INTERFACE ITF_BaseHMIComponent_View EXTENDS ITF_BaseHMILoggerElement_View

METHOD PUBLIC IsValidCommonData : BOOL
VAR_INPUT
END_VAR
END_METHOD

METHOD PUBLIC JoinTheList : INT
VAR_INPUT
	refstList				: REFERENCE TO ST_ListOfElement_HMI;
	iNumberOfParent			: INT; 	//numer rodzica na liście
END_VAR
END_METHOD

METHOD PUBLIC LinkCommonData : BOOL
VAR_INPUT
	stCommonData				: REFERENCE TO ST_BaseCommonData;
END_VAR
END_METHOD

END_INTERFACE

(* stored: Version 1.1.0.1
   Itf ITF_BaseHMIComponent_View: Id {09893359-9aae-0055-210b-9fb2bfb82b06}
   Method IsValidCommonData: Id {3f7a8c5a-8eb8-0328-2fa4-dbdaa99c550b}
   Method JoinTheList: Id {ce02cc1d-c1da-0221-08eb-87e2cdcbb14e}
   Method LinkCommonData: Id {9592f34a-d939-01f0-03b2-89c41fa48d7d} *)
